(* Logix 5000 project; controller ToyPlant Emulate 5570 rev 30.12; software revision 30.00 *)

TASK MainTask (continuous, watchdog 500 ms) : MainProgram

MODULES
   Local : Emulate 5570 (ICP 2, rev 30.12)
      VIRTUAL_INPUTS : vendor 1 type 0 code 15 (ICP 3, rev 1.1, Output RPI 50 ms)
END_MODULES

PROGRAM MainProgram   (* main routine MainRoutine *)
VAR
   A3 : BOOL;
   A3_posinicial : BOOL;
   A4 : BOOL;
   A4_posinicial : BOOL;
   A5 : BOOL;
   A5_posinicial : BOOL;
   A6 : BOOL;
   A6_posinicial : BOOL;
   A7 : BOOL;
   A7_posinicial : BOOL;
   A8 : BOOL;
   A8_posinicial : BOOL;
   A9 : BOOL;
   A9_posinicial : BOOL;
   Action_000 : SFC_ACTION := (Status := 16#0020_0000, PauseTimer := 1);
   Action_001 : SFC_ACTION := (Status := 16#0020_0000, PauseTimer := 1);
   Action_002 : SFC_ACTION := (Status := 16#0020_0000, PauseTimer := 1);
   Action_003 : SFC_ACTION := (Status := 16#0020_0000, PauseTimer := 1);
   Action_004 : SFC_ACTION := (Status := 16#0020_0000, PauseTimer := 1);
   Action_005 : SFC_ACTION := (Status := 16#0020_0000, PauseTimer := 1);
   Action_009 : SFC_ACTION := (Status := 16#0020_0000, PauseTimer := 1);
   Action_010 : SFC_ACTION := (Status := 16#0020_0000, PauseTimer := 1);
   Action_011 : SFC_ACTION := (Status := 16#0020_0000, PauseTimer := 1);
   Action_012 : SFC_ACTION := (Status := 16#0020_0000, PauseTimer := 1);
   Action_013 : SFC_ACTION := (Status := 16#0020_0000, PauseTimer := 1);
   Action_014 : SFC_ACTION := (Status := 16#0020_0000, PauseTimer := 1);
   Action_015 : SFC_ACTION := (Status := 16#0020_0000, PauseTimer := 1);
   Action_016 : SFC_ACTION := (Status := 16#0020_0000, PauseTimer := 1);
   Action_017 : SFC_ACTION := (Status := 16#0020_0000, PauseTimer := 1);
   Action_018 : SFC_ACTION := (Status := 16#0020_0000, PauseTimer := 1);
   Action_019 : SFC_ACTION := (Status := 16#0020_0000, PauseTimer := 1);
   Action_020 : SFC_ACTION := (Status := 16#0020_0000, PauseTimer := 1, Count := 1);
   Action_021 : SFC_ACTION := (Status := 16#c020_0000, A := 1, Q := 1, PauseTimer := 1, Count := 2);
   Action_022 : SFC_ACTION := (Status := 16#0020_0000, PauseTimer := 1, Count := 1);
   Action_023 : SFC_ACTION := (Status := 16#0020_0000, PauseTimer := 1, Count := 1);
   Action_024 : SFC_ACTION := (Status := 16#0020_0000, PauseTimer := 1, Count := 1);
   Action_025 : SFC_ACTION := (Status := 16#0020_0000, PauseTimer := 1, Count := 1);
   Action_026 : SFC_ACTION := (Status := 16#0020_0000, PauseTimer := 1, Count := 1);
   Action_027 : SFC_ACTION := (Status := 16#0020_0000, PauseTimer := 1, Count := 1);
   Action_028 : SFC_ACTION := (Status := 16#0020_0000, PauseTimer := 1, Count := 1);
   AP2 : BOOL;
   AP3 : BOOL;
   banda_1 : DINT;
   Distribucionbandas : BOOL;
   Empaquet : BOOL;
   Enciende : BOOL;
   Ensamble : BOOL;
   R1 : BOOL;
   R2 : BOOL;
   R3 : BOOL;
   s10 : BOOL;
   s6 : BOOL;
   s7 : BOOL;
   s9 : BOOL;
   sensor_detect_barco : BOOL;
   sensor_detect_casa : BOOL;
   sensor_detect_moto : BOOL;
   Servo_posicion_final : BOOL;
   Servo_posicion_media : BOOL;
   si1 : BOOL;
   si2 : BOOL;
   si3 : BOOL;
   Start_banda_1 : DINT;
   Start_banda_2 : BOOL;
   Start_banda_3 : BOOL;
   start_empaquetamiento : BOOL;
   StartEnsamble : ALIAS FOR Local:3:I.Data[1].0;
   Step_000 : SFC_STEP := (Status := 16#0020_0000, PauseTimer := 1);
   Step_001 : SFC_STEP := (Status := 16#0020_0000, PauseTimer := 1);
   Step_002 : SFC_STEP := (Status := 16#0020_0000, PauseTimer := 1);
   Step_003 : SFC_STEP := (Status := 16#0020_0000, PauseTimer := 1);
   Step_004 : SFC_STEP := (Status := 16#0020_0000, PauseTimer := 1);
   Step_005 : SFC_STEP := (Status := 16#0020_0000, PauseTimer := 1);
   Step_006 : SFC_STEP := (Status := 16#0020_0000, PauseTimer := 1);   // Ensamble Barco
   Step_007 : SFC_STEP := (Status := 16#0020_0000, PauseTimer := 1);
   Step_008 : SFC_STEP := (Status := 16#0020_0000, PauseTimer := 1);
   Step_009 : SFC_STEP := (Status := 16#0020_0000, PauseTimer := 1);
   Step_010 : SFC_STEP := (Status := 16#0020_0000, PauseTimer := 1);
   Step_011 : SFC_STEP := (Status := 16#0020_0000, PauseTimer := 1, PRE := 2000);
   Step_012 : SFC_STEP := (Status := 16#0020_0000, PauseTimer := 1, PRE := 7000);
   Step_013 : SFC_STEP := (Status := 16#0020_0000, PauseTimer := 1);
   Step_014 : SFC_STEP := (Status := 16#0020_0000, PauseTimer := 1);
   Step_015 : SFC_STEP := (Status := 16#0020_0000, PauseTimer := 1);
   Step_016 : SFC_STEP := (Status := 16#0020_0000, PauseTimer := 1);   // Inicio de ensamble casa
   Step_017 : SFC_STEP := (Status := 16#0020_0000, PauseTimer := 1, PRE := 4000);
   Step_018 : SFC_STEP := (Status := 16#0020_0000, PauseTimer := 1, PRE := 3000);
   Step_019 : SFC_STEP := (Status := 16#a820_0201, X := 1, SA := 1, DN := 1, PauseTimer := 1, T := 31632, TMax := 31632, Count := 2);
   Step_020 : SFC_STEP := (Status := 16#0820_0001, DN := 1, PauseTimer := 1, T := 2120, TMax := 2120, Count := 1);
   Step_021 : SFC_STEP := (Status := 16#0820_0001, DN := 1, PauseTimer := 1, T := 6321, TMax := 6321, Count := 1);
   Step_022 : SFC_STEP := (Status := 16#0820_0001, DN := 1, PauseTimer := 1, T := 741, TMax := 741, Count := 1);
   Step_023 : SFC_STEP := (Status := 16#0820_0001, DN := 1, PauseTimer := 1, T := 933, TMax := 933, Count := 1);
   Step_024 : SFC_STEP := (Status := 16#0820_0001, DN := 1, PauseTimer := 1, T := 527, TMax := 527, Count := 1);
   Stop_banda_1 : BOOL;
   Stop_banda_2 : BOOL;
   Stop_banda_3 : BOOL;
   TimerChasis : FBD_TIMER := (TimerEnable := 1, PRE := 700, ACC := 720, EN := 1, DN := 1);
   TimerPuertaAbierta : FBD_TIMER := (TimerEnable := 1, PRE := 900, ACC := 912, EN := 1, DN := 1);
   TimerPuertaCerrada : FBD_TIMER := (TimerEnable := 1, PRE := 500, ACC := 500, EN := 1, DN := 1);
   Tran_000 : BOOL;
   Tran_001 : BOOL;
   Tran_002 : BOOL;
   Tran_003 : BOOL;
   Tran_004 : BOOL;
   Tran_005 : BOOL;
   Tran_006 : BOOL;
   Tran_007 : BOOL;
   Tran_008 : BOOL;
   Tran_009 : BOOL;
   Tran_010 : BOOL;
   Tran_011 : BOOL;
   Tran_012 : BOOL;
   Tran_013 : BOOL;
   Tran_014 : BOOL;
   Tran_015 : BOOL;
   Tran_016 : BOOL;
   Tran_017 : BOOL;
   Tran_018 : BOOL;
   Tran_019 : BOOL;
   Tran_020 : BOOL := 1;
   Tran_021 : BOOL := 1;
   Tran_022 : BOOL := 1;
   Tran_023 : BOOL := 1;
   Tran_024 : BOOL := 1;
END_VAR
VAR_OUTPUT
   CerrarPuertaMoto : BOOL := 1; {access Read Only}
   Chasis_0 : BOOL := 1;
   Chasis_1 : BOOL := 1;
   RuedaDelantera_0 : BOOL := 1;
   RuedaDelantera_1 : BOOL := 1;
   RuedaDelantera_2 : BOOL := 1;
   RuedaTrasera_0 : BOOL := 1;
   RuedaTrasera_1 : BOOL := 1;
   RuedaTrasera_2 : BOOL := 1;
END_VAR
VAR_INPUT
   Sensor_RuedaDelantera1 : BOOL;
   Sensor_RuedaDelantera2 : BOOL;
   Sensor_RuedaTrasera1 : BOOL;
   Sensor_RuedaTrasera2 : BOOL;
   SensorChasis : BOOL;
END_VAR

ROUTINE Barco   (* sequential function chart *)
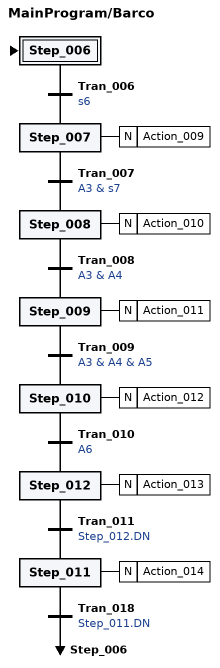
   INITIAL_STEP Step_006:
   END_STEP
   TRANSITION Tran_006 FROM Step_006 TO Step_007
      := s6
   END_TRANSITION
   STEP Step_007:
      ACTION Action_009 (N):
         A3 := 1;
      END_ACTION
   END_STEP
   TRANSITION Tran_007 FROM Step_007 TO Step_008
      := A3 & s7
   END_TRANSITION
   STEP Step_008:
      ACTION Action_010 (N):
         A4:=1;
      END_ACTION
   END_STEP
   TRANSITION Tran_008 FROM Step_008 TO Step_009
      := A3 & A4
   END_TRANSITION
   STEP Step_009:
      ACTION Action_011 (N):
         A5 :=1;
      END_ACTION
   END_STEP
   TRANSITION Tran_009 FROM Step_009 TO Step_010
      := A3 & A4 & A5
         
   END_TRANSITION
   STEP Step_010:
      ACTION Action_012 (N):
         A6 := 1;
      END_ACTION
   END_STEP
   TRANSITION Tran_010 FROM Step_010 TO Step_012
      := A6
         
   END_TRANSITION
   STEP Step_012:
      ACTION Action_013 (N):
         A3_posinicial :=1;
         A4_posinicial :=1;
         A5_posinicial :=1;
         A6_posinicial :=1;
      END_ACTION
   END_STEP
   TRANSITION Tran_011 FROM Step_012 TO Step_011
      := Step_012.DN
         
   END_TRANSITION
   STEP Step_011:
      ACTION Action_014 (N):
         AP2:=1;
      END_ACTION
   END_STEP
   TRANSITION Tran_018 FROM Step_011 TO Step_006
      := Step_011.DN
         
   END_TRANSITION
END_ROUTINE

ROUTINE Casa   (* sequential function chart *)
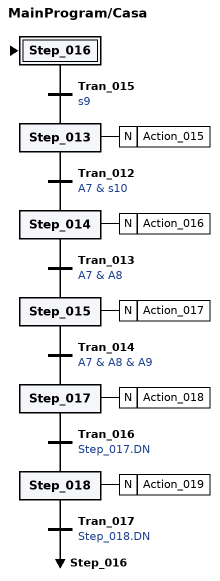
   INITIAL_STEP Step_016:
   END_STEP
   TRANSITION Tran_015 FROM Step_016 TO Step_013
      := s9
   END_TRANSITION
   STEP Step_013:
      ACTION Action_015 (N):
         A7 :=1;
      END_ACTION
   END_STEP
   TRANSITION Tran_012 FROM Step_013 TO Step_014
      := A7 & s10
   END_TRANSITION
   STEP Step_014:
      ACTION Action_016 (N):
         A8 := 1;
      END_ACTION
   END_STEP
   TRANSITION Tran_013 FROM Step_014 TO Step_015
      := A7 & A8
   END_TRANSITION
   STEP Step_015:
      ACTION Action_017 (N):
         A9 :=1;
      END_ACTION
   END_STEP
   TRANSITION Tran_014 FROM Step_015 TO Step_017
      := A7 & A8 & A9
   END_TRANSITION
   STEP Step_017:
      ACTION Action_018 (N):
         A7_posinicial :=1;
         A8_posinicial :=1;
         A9_posinicial :=1;
      END_ACTION
   END_STEP
   TRANSITION Tran_016 FROM Step_017 TO Step_018
      := Step_017.DN
         
   END_TRANSITION
   STEP Step_018:
      ACTION Action_019 (N):
         AP3 :=1 ;
      END_ACTION
   END_STEP
   TRANSITION Tran_017 FROM Step_018 TO Step_016
      := Step_018.DN
         
   END_TRANSITION
END_ROUTINE

ROUTINE Distribucion_de_caja_en_bandas   (* sequential function chart *)
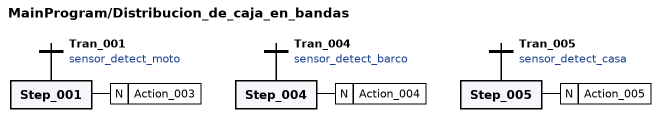
   TRANSITION Tran_001 FROM () TO Step_001
      := sensor_detect_moto
   END_TRANSITION
   TRANSITION Tran_004 FROM () TO Step_004
      := sensor_detect_barco
         
   END_TRANSITION
   TRANSITION Tran_005 FROM () TO Step_005
      := sensor_detect_casa
         
   END_TRANSITION
   STEP Step_001:
      ACTION Action_003 (N):
         Start_banda_1 :=1;
         Stop_banda_2 :=1;
         Stop_banda_3 :=1;
      END_ACTION
   END_STEP
   STEP Step_005:
      ACTION Action_005 (N):
         Start_banda_3 :=1;
         Stop_banda_2 :=1;
         Stop_banda_1 :=1;
         Servo_posicion_final:=1;
      END_ACTION
   END_STEP
   STEP Step_004:
      ACTION Action_004 (N):
         Start_banda_2 :=1;
         Stop_banda_3 :=1;
         Stop_banda_1 :=1;
         Servo_posicion_media:=1;
      END_ACTION
   END_STEP
END_ROUTINE

ROUTINE Empaquetamiento   (* sequential function chart *)
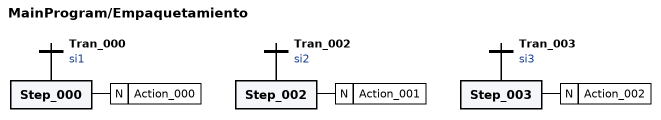
   TRANSITION Tran_000 FROM () TO Step_000
      := si1
   END_TRANSITION
   TRANSITION Tran_002 FROM () TO Step_002
      := si2
   END_TRANSITION
   TRANSITION Tran_003 FROM () TO Step_003
      := si3
   END_TRANSITION
   STEP Step_000:
      ACTION Action_000 (N):
         R1:=1;
      END_ACTION
   END_STEP
   STEP Step_002:
      ACTION Action_001 (N):
         R2:=1;
      END_ACTION
   END_STEP
   STEP Step_003:
      ACTION Action_002 (N):
         R3:=1;
      END_ACTION
   END_STEP
END_ROUTINE

ROUTINE Mainprogram_Ladder   (* ladder *)
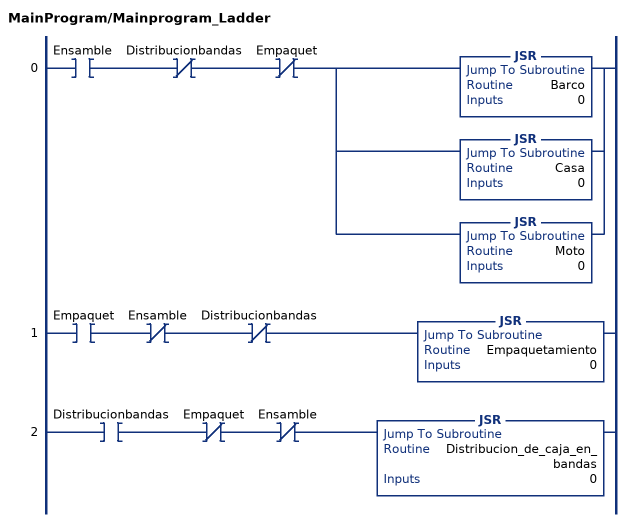
   0: XIC(Ensamble)XIO(Distribucionbandas)XIO(Empaquet)[JSR(Barco,0) ,JSR(Casa,0) ,JSR(Moto,0) ];
   1: XIC(Empaquet)XIO(Ensamble)XIO(Distribucionbandas)JSR(Empaquetamiento,0);
   2: XIC(Distribucionbandas)XIO(Empaquet)XIO(Ensamble)JSR(Distribucion_de_caja_en_bandas,0);
END_ROUTINE

ROUTINE MainRoutine   (* sequential function chart *)
END_ROUTINE

ROUTINE Moto   (* sequential function chart *)
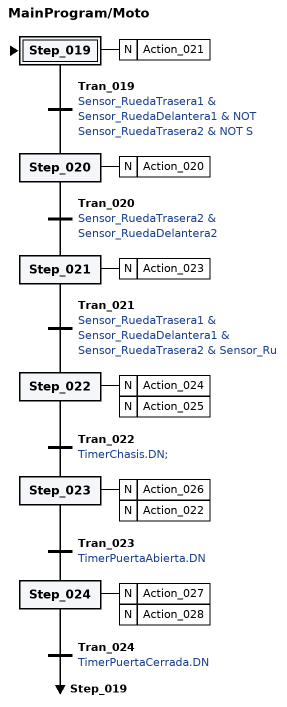
   INITIAL_STEP Step_019:
      ACTION Action_021 (N):
         CerrarPuertaMoto := 1;
      END_ACTION
   END_STEP
   TRANSITION Tran_019 FROM Step_019 TO Step_020
      := Sensor_RuedaTrasera1 & Sensor_RuedaDelantera1 & NOT Sensor_RuedaTrasera2 & NOT Sensor_RuedaDelantera2 & CerrarPuertaMoto
         
   END_TRANSITION
   STEP Step_020:
      ACTION Action_020 (N):
         RuedaDelantera_1 := 1;
         RuedaTrasera_1 := 1;
      END_ACTION
   END_STEP
   TRANSITION Tran_020 FROM Step_020 TO Step_021
      := Sensor_RuedaTrasera2 & Sensor_RuedaDelantera2
         
   END_TRANSITION
   STEP Step_021:
      ACTION Action_023 (N):
         RuedaTrasera_0 := 1;
         RuedaDelantera_0 := 1;
      END_ACTION
   END_STEP
   TRANSITION Tran_021 FROM Step_021 TO Step_022
      := Sensor_RuedaTrasera1 & Sensor_RuedaDelantera1 & Sensor_RuedaTrasera2 & Sensor_RuedaDelantera2 & SensorChasis
   END_TRANSITION
   STEP Step_022:
      ACTION Action_024 (N):
         Chasis_1 := 1;
      END_ACTION
      ACTION Action_025 (N):
         TimerChasis.TimerEnable := 1;
         TONR(TimerChasis);
         TimerChasis.PRE := 700;
         
      END_ACTION
   END_STEP
   TRANSITION Tran_022 FROM Step_022 TO Step_023
      := TimerChasis.DN;
   END_TRANSITION
   STEP Step_023:
      ACTION Action_026 (N):
         RuedaTrasera_2 := 1;
         RuedaDelantera_2 := 1;
      END_ACTION
      ACTION Action_022 (N):
         TimerPuertaAbierta.TimerEnable := 1;
         TONR(TimerPuertaAbierta);
         TimerPuertaAbierta.PRE := 900;
         
      END_ACTION
   END_STEP
   TRANSITION Tran_023 FROM Step_023 TO Step_024
      := TimerPuertaAbierta.DN
   END_TRANSITION
   STEP Step_024:
      ACTION Action_027 (N):
         CerrarPuertaMoto := 0;
         RuedaTrasera_0 := 1;
         RuedaDelantera_0 := 1;
         Chasis_0 :=1;
      END_ACTION
      ACTION Action_028 (N):
         TimerPuertaCerrada.TimerEnable := 1;
         TONR(TimerPuertaCerrada);
         TimerPuertaCerrada.PRE := 500;
         
      END_ACTION
   END_STEP
   TRANSITION Tran_024 FROM Step_024 TO Step_019
      := TimerPuertaCerrada.DN
   END_TRANSITION
END_ROUTINE
END_PROGRAM
